// TIA Portal project "FactoryIO_Template_S7-1200_V15_V18" (V18)
// Vorlageprojekt für das Buch mit Zielsystem S7-1200

(* hardware
DEVICE "S7-1200-Station_1"  S7-1200 Station
   slot 0: "Baugruppenträger_0"  Rack  V1.0
   slot 1: "PLC_1"  CPU 1214C DC/DC/DC  6ES7 214-1AG40-0XB0  V4.6
*)

// ===== PLC "PLC_1"  CPU 1214C DC/DC/DC =====

VAR_GLOBAL   // PLC tag table "Standard-Variablentabelle"
   "START BUT" AT %I0.0 : Bool;
   "STOP BUT" AT %I0.1 : Bool;
   "SENSOR 1" AT %I0.2 : Bool;
   "SENSOR 2" AT %I0.3 : Bool;
   "SENSOR 3" AT %I0.4 : Bool;
   "PLAT. LIM. SENSOR" AT %I0.5 : Bool;
   "ASAN. LIM. SENSOR" AT %I0.6 : Bool;
   "KONVEYOR 1" AT %Q0.0 : Bool;
   "KONVEYOR 2" AT %Q0.1 : Bool;
   "PLAT. ILERI" AT %Q0.2 : Bool;
   "PLAT. DONDURME" AT %Q0.3 : Bool;
   "ASAN. ILERI" AT %Q0.4 : Bool;
   "ASAN. YUKARI" AT %Q0.5 : Bool;
   "PLAT. DONUS SENSORU" AT %I0.7 : Bool;
END_VAR

// folder: System blocks/Program resources

DATA_BLOCK "TIMER 1"   // DB1
{ S7_Optimized_Access := 'TRUE' }
AUTHOR : Simatic
FAMILY : IEC
NAME : IEC_TMR
VERSION : 1.0
// stored: InstanceOfName IEC_TIMER
"IEC_TIMER"
BEGIN
END_DATA_BLOCK

// folder: (top level)

FUNCTION "MHJ-PLC-Lab-Function-S71200" : Void   // FC9000, SCL
{ S7_Optimized_Access := 'TRUE' }
VERSION : 0.1
   VAR_TEMP
      rdTimeReturn : Int;
      outputTime : DTL;
      SyncVal : Byte;
      forVal : Int;
      forVal_2 : Int;
      Value : Byte;
   END_VAR
   VAR CONSTANT
      CompVal : Byte := 16#34;
      Value_01 : Byte := 16#11;
      Value_01_DW : DWord := 16#A165_D992;
      Value_02_DW : DWord := 16#58BE_4401;
   END_VAR
BEGIN

   #Value:=PEEK(area := 16#82,
        dbNumber := 0,
        byteOffset := 511);
   #Value := #Value + 1;

   POKE(area := 16#82,
        dbNumber := 0,
        byteOffset := 511,
        value := #Value);

   POKE(area:=16#81,
        dbNumber:=0,
        byteOffset:=1016,
        value:=#Value_01_DW);
   POKE(area := 16#81,
        dbNumber := 0,
        byteOffset := 1020,
        value := #Value_02_DW);

   POKE(area := 16#81,
        dbNumber := 0,
        byteOffset := 511,
        value := B#16#00);

   FOR #forVal := 0 TO 120 DO
       FOR #forVal_2:=0 TO 10 DO
           #rdTimeReturn:=RD_SYS_T(#outputTime);
           #rdTimeReturn := WR_SYS_T(#outputTime);
           #rdTimeReturn := RD_SYS_T(#outputTime);
           #rdTimeReturn := WR_SYS_T(#outputTime);
       END_FOR;
       #SyncVal:= PEEK(area := 16#81,
                      dbNumber := 0,
                      byteOffset := 511);
       IF #SyncVal = #CompVal THEN
          GOTO M_1;
       END_IF;
   END_FOR;
   RETURN;

   M_1:
   POKE(area := 16#81,
        dbNumber := 0,
        byteOffset := 511,
        value := B#16#0);
END_FUNCTION

ORGANIZATION_BLOCK "Main"   // OB1, LAD, ProgramCycle
TITLE = "Main Program Sweep (Cycle)"
{ S7_Optimized_Access := 'TRUE' }
VERSION : 0.1
   VAR_INPUT
      Initial_Call : Bool;   // Initial call of this OB
      Remanence : Bool;   // =True, if remanent data are available
   END_VAR
BEGIN

REGION Network 1: Konnektierungsbaustein für PLC-Lab / KÜTÜPHANE BLOĞU
   // Im Netzwerk 1 wird der Konnektierungsbaustein für PLC-Lab aufgerufen.
   // Dieser Aufruf darf nicht entfernt werden!
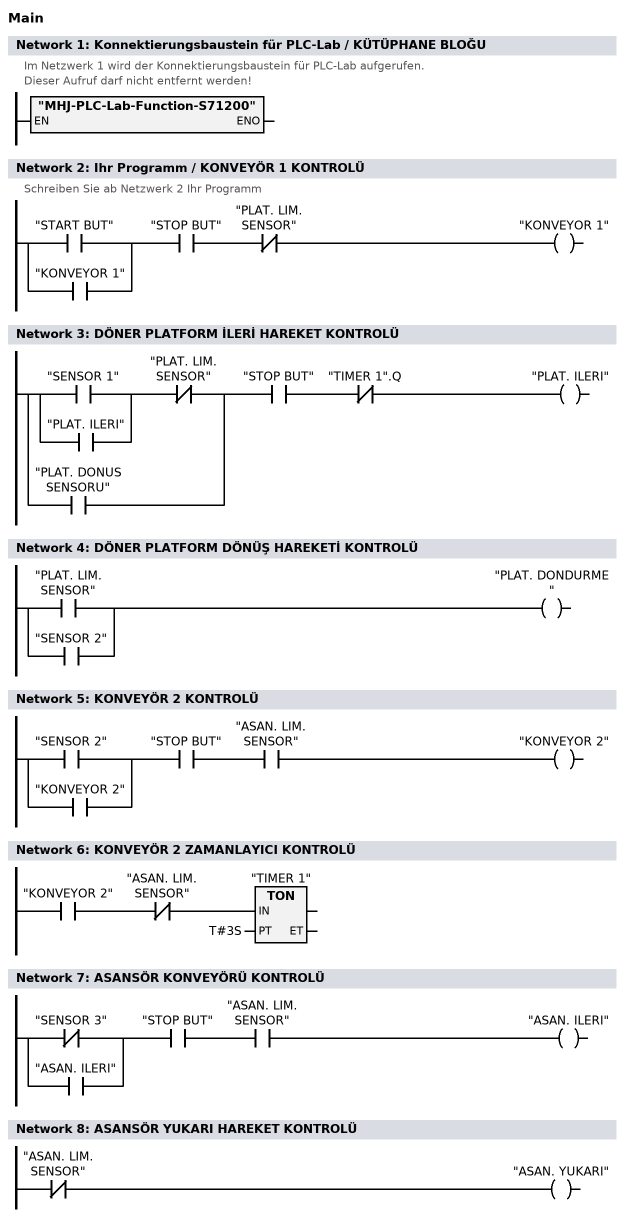
   RUNG wire#powerrail
      "MHJ-PLC-Lab-Function-S71200"()
   END_RUNG
   // the same network as SCL:
   "MHJ-PLC-Lab-Function-S71200"();
END_REGION

REGION Network 2: Ihr Programm / KONVEYÖR 1 KONTROLÜ
   // Schreiben Sie ab Netzwerk 2 Ihr Programm
   RUNG wire#powerrail
      Contact( "START BUT" )
      wire#w1
      Contact( "STOP BUT" )
      I_Contact( "PLAT. LIM. SENSOR" )
      Coil( "KONVEYOR 1" )
   END_RUNG
   RUNG wire#powerrail
      Contact( "KONVEYOR 1" )
   END_RUNG wire#w1
   // the same network as SCL:
   "KONVEYOR 1" := ("START BUT" OR "KONVEYOR 1") AND "STOP BUT" AND NOT "PLAT. LIM. SENSOR";
END_REGION

REGION Network 3: DÖNER PLATFORM İLERİ HAREKET KONTROLÜ
   RUNG wire#powerrail
      Contact( "SENSOR 1" )
      wire#w1
      I_Contact( "PLAT. LIM. SENSOR" )
      wire#w2
      Contact( "STOP BUT" )
      I_Contact( "TIMER 1".Q )
      Coil( "PLAT. ILERI" )
   END_RUNG
   RUNG wire#powerrail
      Contact( "PLAT. ILERI" )
   END_RUNG wire#w1
   RUNG wire#powerrail
      Contact( "PLAT. DONUS SENSORU" )
   END_RUNG wire#w2
   // the same network as SCL:
   "PLAT. ILERI" := ((("SENSOR 1" OR "PLAT. ILERI") AND NOT "PLAT. LIM. SENSOR") OR "PLAT. DONUS SENSORU") AND "STOP BUT" AND NOT "TIMER 1".Q;
END_REGION

REGION Network 4: DÖNER PLATFORM DÖNÜŞ HAREKETİ KONTROLÜ
   RUNG wire#powerrail
      Contact( "PLAT. LIM. SENSOR" )
      wire#w1
      Coil( "PLAT. DONDURME" )
   END_RUNG
   RUNG wire#powerrail
      Contact( "SENSOR 2" )
   END_RUNG wire#w1
   // the same network as SCL:
   "PLAT. DONDURME" := "PLAT. LIM. SENSOR" OR "SENSOR 2";
END_REGION

REGION Network 5: KONVEYÖR 2 KONTROLÜ
   RUNG wire#powerrail
      Contact( "SENSOR 2" )
      wire#w1
      Contact( "STOP BUT" )
      Contact( "ASAN. LIM. SENSOR" )
      Coil( "KONVEYOR 2" )
   END_RUNG
   RUNG wire#powerrail
      Contact( "KONVEYOR 2" )
   END_RUNG wire#w1
   // the same network as SCL:
   "KONVEYOR 2" := ("SENSOR 2" OR "KONVEYOR 2") AND "STOP BUT" AND "ASAN. LIM. SENSOR";
END_REGION

REGION Network 6: KONVEYÖR 2 ZAMANLAYICI KONTROLÜ
   "TIMER 1".TON(IN := "KONVEYOR 2" AND NOT "ASAN. LIM. SENSOR", PT := T#3S);
END_REGION

REGION Network 7: ASANSÖR KONVEYÖRÜ KONTROLÜ
   RUNG wire#powerrail
      I_Contact( "SENSOR 3" )
      wire#w1
      Contact( "STOP BUT" )
      Contact( "ASAN. LIM. SENSOR" )
      Coil( "ASAN. ILERI" )
   END_RUNG
   RUNG wire#powerrail
      Contact( "ASAN. ILERI" )
   END_RUNG wire#w1
   // the same network as SCL:
   "ASAN. ILERI" := (NOT "SENSOR 3" OR "ASAN. ILERI") AND "STOP BUT" AND "ASAN. LIM. SENSOR";
END_REGION

REGION Network 8: ASANSÖR YUKARI HAREKET KONTROLÜ
   RUNG wire#powerrail
      I_Contact( "ASAN. LIM. SENSOR" )
      Coil( "ASAN. YUKARI" )
   END_RUNG
   // the same network as SCL:
   "ASAN. YUKARI" := NOT "ASAN. LIM. SENSOR";
END_REGION
END_ORGANIZATION_BLOCK